PROGRAM MAIN
VAR

END_VAR


AssignInsOuts();

HMI_Functions();

CASE GVL_HMI.ProgramSelect OF
	1:
		Part1();
	2:
		Part2();
	3:
		Part3();
END_CASE

END_PROGRAM

(* stored: Version 1.1.0.1
   POU MAIN: Id {3a9dacf3-edac-469c-b94b-870f261e6860}, SpecialFunc None *)
